// TIA Portal V16 export
// export: Created 2024-09-05T17:40:15.1498979Z, ExportSetting WithDefaults, DisplayName Totally Integrated Automation Portal, DisplayVersion V16 Update 6, DisplayName TIA Portal Version Control Interface, DisplayVersion V16 Update 2, DisplayName TIA Portal Openness, DisplayVersion V16 Update 6, DisplayName STEP 7 Professional, DisplayVersion V16 Update 6, DisplayName STEP 7 Safety, DisplayVersion V16, DisplayName WinCC Advanced, DisplayVersion V16 Update 6
TYPE "udtModes"
// stored: IsFailsafeCompliant false
   STRUCT
      activeMode : Int;
      switch : Struct
         auto : Bool;
         poloautomaActivated : Bool;
         stepModeActivated : Bool;
      END_STRUCT;
      button : Struct
         basic : Struct
            request : Struct
               button : Bool;
               visibility : Bool;
            END_STRUCT;
         END_STRUCT;
         auto : Struct
            startRequest : Struct
               button : Bool;
               visibility : Bool;
            END_STRUCT;
            stopRequest : Struct
               button : Bool;
               visibility : Bool;
            END_STRUCT;
            emptyRequest : Struct
               button : Bool;
               visibility : Bool;
            END_STRUCT;
         END_STRUCT;
         "step" : Bool;
         poloautomatStart : Array[0..25] of Bool;
      END_STRUCT;
      modeChanged : Bool;
      autoStatus : Struct
         stopping : Bool;
         stopped : Bool;
         emptying : Bool;
         empty : Bool;
      END_STRUCT;
      StationNrForPoloautomat_step : Int;
   END_STRUCT;
END_TYPE
